// TIA Portal V17 export
// export: Created 2024-09-02T12:50:30.5171932Z, ExportSetting WithDefaults, DisplayName Totally Integrated Automation Portal, DisplayVersion V17, DisplayName TIA Portal Openness, DisplayVersion V17, DisplayName TIA Portal Version Control Interface, DisplayVersion V17, DisplayName STEP 7 Professional, DisplayVersion V17, DisplayName STEP 7 Safety, DisplayVersion V17, DisplayName WinCC Professional, DisplayVersion V17
TYPE "type_CognexVsOut"
// stored: IsFailsafeCompliant false
   STRUCT
      Ansteuerung { ExternalWritable := 'False'} : Struct   // Ansteuerung / Control
         Trigger_enable { ExternalWritable := 'False'} : Bool;   // Aufnamesteuerung: Trigger enable / Recording Status: Trigger enable
         Trigger { ExternalWritable := 'False'} : Bool;   // Aufnamesteuerung: Trigger / Recording Status: Trigger
         Res02 { ExternalWritable := 'False'} : Bool;   // Aufnamesteuerung: / Record control:
         Res03 { ExternalWritable := 'False'} : Bool;   // Aufnamesteuerung: / Record control:
         Res04 { ExternalWritable := 'False'} : Bool;   // Aufnamesteuerung: / Record control:
         Res05 { ExternalWritable := 'False'} : Bool;   // Aufnamesteuerung: / Record control:
         Res06 { ExternalWritable := 'False'} : Bool;   // Aufnamesteuerung: / Record control:
         Set_Offline { ExternalWritable := 'False'} : Bool;   // Aufnahmesteurung: Set offline / Recording status: Set offline
         Buffer_Results_Enable { ExternalWritable := 'False'} : Bool;   // Inspektionssteuerung: Buffer Results Enable / Inspection Control: Buffer Results Enable
         Inspection_Results_Ack { ExternalWritable := 'False'} : Bool;   // Inspektionssteuerung: Inspection Results Acknowledge / Inspection Control: Inspection Results Acknowledge
         Res11 { ExternalWritable := 'False'} : Bool;   // Inspektionssteuerung: / Inspection control:
         Res12 { ExternalWritable := 'False'} : Bool;   // Inspektionssteuerung: / Inspection control:
         Res13 { ExternalWritable := 'False'} : Bool;   // Inspektionssteuerung: / Inspection control:
         Res14 { ExternalWritable := 'False'} : Bool;   // Inspektionssteuerung: / Inspection control:
         Res15 { ExternalWritable := 'False'} : Bool;   // Inspektionssteuerung: / Inspection control:
         Res16 { ExternalWritable := 'False'} : Bool;   // Inspektionssteuerung: / Inspection control:
         Set_Job_No { ExternalWritable := 'False'} : Byte;   // Parametersatz: Set Job Number / Parameter set: Set Job Number
         Softevent { ExternalWritable := 'False'} : Byte;   // Softevent / soft event
      END_STRUCT;
      Benutzerdaten { ExternalWritable := 'False'} : Struct   // Benutzerdaten (ab Byte 4) / User name (ab Byte 4)
         Ausfuehrungskennung { ExternalWritable := 'False'} : Struct   // Kennung / ID
            Kennung01 { ExternalWritable := 'False'} : Char;   // Kennung für die Ausführungsart des IBV-Systems / Identifier for the type of implementation of the IBV system
            Kennung02 { ExternalWritable := 'False'} : Char;   // Kennung für die Ausführungsart des IBV-Systems / Identifier for the type of implementation of the IBV system
         END_STRUCT;
         Zeitstempel { ExternalWritable := 'False'} : Struct   // Zeitstempel / Time stamp
            Jahr_0 { ExternalWritable := 'False'} : Char;   // Jahr im Format JJJJ (4. Stelle) / Year in format YYYY (4th position)
            Jahr_1 { ExternalWritable := 'False'} : Char;   // Jahr im Format JJJJ (3. Stelle) / Year in format YYYY (3rd position)
            Jahr_2 { ExternalWritable := 'False'} : Char;   // Jahr im Format JJJJ (2. Stelle) / Year in format YYYY (2nd position)
            Jahr_3 { ExternalWritable := 'False'} : Char;   // Jahr im Format JJJJ (1. Stelle) / Year in format YYYY (1st position)
            Mon_0 { ExternalWritable := 'False'} : Char;   // Monat im Format MM (2. Stelle) / Month in MM format (2 st digit)
            Mon_1 { ExternalWritable := 'False'} : Char;   // Monat im Format MM (1. Stelle) / Month in MM format (1st digit)
            Tag_0 { ExternalWritable := 'False'} : Char;   // Tag im Format TT (2. Stelle) / Tag in TT format (2st digit)
            Tag_1 { ExternalWritable := 'False'} : Char;   // Tag im Format TT (1. Stelle) / Tag in TT format (1st digit)
            Std_0 { ExternalWritable := 'False'} : Char;   // Stunden im Format hh (2. Stelle) / Hours in hh format (2nd digit)
            Std_1 { ExternalWritable := 'False'} : Char;   // Stunden im Format hh (1. Stelle) / Hours in hh format (1st digit)
            Min_0 { ExternalWritable := 'False'} : Char;   // Minuten im Format mm (2. Stelle) / Minutes in mm format (1st digit)
            Min_1 { ExternalWritable := 'False'} : Char;   // Minuten im Format mm (1. Stelle) / Minutes in mm format (1st digit)
            Sek_0 { ExternalWritable := 'False'} : Char;   // Sekunden im Format ss (2. Stelle) / Seconds in ss format (2 position)
            Sek_1 { ExternalWritable := 'False'} : Char;   // Sekunden im Format ss (1. Stelle) / Seconds in ss format (1 position)
         END_STRUCT;
         Daten { ExternalWritable := 'False'} : Struct   // Daten / Data
            StationsNr { ExternalWritable := 'False'} : Array[1..6] of Char;   // Adr.16
            KameraNr { ExternalWritable := 'False'} : Array[1..2] of Char;   // Adr.22
            PID { ExternalWritable := 'False'} : Array[1..30] of Char;   // Adr.24
            MotNr { ExternalWritable := 'False'} : Array[1..12] of Char;   // Adr.54
            ProgrammNr { ExternalWritable := 'False'} : Array[1..2] of Char;   // Adr.66
            ErweiterteDaten { ExternalWritable := 'False'} : Array[1..30] of Char;   // Adr.68
            Res { ExternalWritable := 'False'} : Array[98..127] of Char;   // Adr.98
         END_STRUCT;
      END_STRUCT;
   END_STRUCT;
END_TYPE
